// TIA Portal project "VISU_Umsetzer+Sauggreifer_Template" (V14)

(* hardware
DEVICE "S7300/ET200M-Station_1"  S7-300 station
   slot 0: "Profilschiene_0"  Rail  6ES7 390-1***0-0AA0
   slot 2: "PLC_1"  CPU 315-2 PN/DP  6ES7 315-2EH13-0AB0  V2.6
      slot 1: "MPI/DP-Schnittstelle_1"  X1
      slot 2: "PROFINET-Schnittstelle_1"  PN-IO
         slot 1: "Port_1"  Port
*)

// ===== PLC "PLC_1"  CPU 315-2 PN/DP =====

VAR_GLOBAL   // PLC tag table "Standard-Variablentabelle"
   "POS_X_PLUS" AT %I10.3 : Bool;   // Greifer bei Position X+
   "POS_X_MIDDLE" AT %I10.4 : Bool;   // Greifer bei Position X Mitte
   "POS_X_MINUS" AT %I10.5 : Bool;   // Greifer bei Position X-
   "POS_Z_PLUS" AT %I10.6 : Bool;   // Greifer bei Position Z+
   "POS_Z_MINUS" AT %I10.7 : Bool;   // Greifer bei Position Z-
   "STORAGE_ENGAGED" AT %I11.0 : Bool;   // Ablageplatz belegt
   "BELT1_ENGAGED" AT %I11.3 : Bool;   // Förderband 1 belegt
   "BELT2_ENGAGED" AT %I11.4 : Bool;   // Förderband 2 belegt
   "TO_X_PLUS" AT %Q4.0 : Bool;   // Greifer nach X+ fahren
   "TO_X_MINUS" AT %Q4.1 : Bool;   // Greifer nach X- fahren
   "TO_Z_PLUS" AT %Q4.2 : Bool;   // Greifer nach Z+ fahren
   "TO_Z_MINUS" AT %Q4.3 : Bool;   // Greifer nach Z- fahren
   "BELT1_TO_X_PLUS" AT %Q4.4 : Bool;   // Förderband 1 nach X+
   "BELT1_TO_X_MINUS" AT %Q4.5 : Bool;   // Förderband 1 nach X-
   "BELT2_TO_X_PLUS" AT %Q4.6 : Bool;   // Förderband 2 nach X+
   "BELT2_TO_X_MINUS" AT %Q4.7 : Bool;   // Förderband 2 nach X-
   "PUMP_ON" AT %Q5.0 : Bool;   // Greiferpumpe an
   "CONTROL_KEY_1" AT %I11.1 : Bool;   // Bedientaster 1
   "CONTROL_KEY_2" AT %I11.2 : Bool;   // Bedientaster 2
   "INIT_0" AT %M0.0 : Bool;   // 1 - Initschritt 0 abgeschlossen
   "INIT_1" AT %M0.1 : Bool;   // 1 - Initschritt 1 abgeschlossen
   "INIT_2" AT %M0.2 : Bool;   // 1 - Initschritt 2 abgeschlossen
   "STEP" AT %MW2 : Int;
   "RESET(1)" AT %M1.6 : Bool;
   "Trig_ContrKey1" AT %M0.3 : Bool;   // 1 - Pos Flanke
   "Trig_Step_1" AT %M0.6 : Bool;   // 1 - Pos Flanke
   "Trig_ContrKey2" AT %M0.4 : Bool;   // 1 - Pos Flanke
   "STORAGE" AT %M1.3 : Bool;   // 1 - Ablage zu Belt 2
   "Trig_Step_2" AT %M0.7 : Bool;   // 1 - Pos Flanke
   "BELT1_BELT2" AT %M1.2 : Bool;
   "BELT1_STORAGE" AT %M1.1 : Bool;
   "Trig_Step_3" AT %M1.0 : Bool;   // 1 - Pos Flanke
   "INC_CHN_A" AT %I10.0 : Bool;   // Inkrementalgeber X-Achse Kanal A
   "INC_CHN_B" AT %I10.1 : Bool;   // Inkrementalgeber X-Achse Kanal B
   "INC_CHN_Z" AT %I10.2 : Bool;   // Inkrementalgeber X-Achse Kanal C
   "X_POSITION" AT %MD1000 : DInt;   // X-Position Greifer
   "Trig_Chan_A" AT %M1.5 : Bool;   // 1 - Pos Flanke
   "Trig_Chan_B" AT %M1.4 : Bool;   // 1 - Pos Flanke
   "INTERN" AT %MW6 : Int;
   "D_INTERN" AT %MD8 : DInt;
END_VAR

DATA_BLOCK "Incremental_DB"   // DB2
{ S7_Optimized_Access := 'FALSE' }
VERSION : 0.1
// stored: InstanceOfName Incremental
"Incremental"
BEGIN
END_DATA_BLOCK

FUNCTION_BLOCK "Incremental"   // FB1, FBD
{ S7_Optimized_Access := 'FALSE' }
VERSION : 0.1
   VAR_INPUT
      KANAL_A : Bool;
      KANAL_B : Bool;
      RESET : Bool;
   END_VAR
   VAR_OUTPUT
      Number : DInt;
   END_VAR
   VAR_TEMP   // added for the SCL form of the ladder/FBD networks
      _w1 : Bool;
   END_VAR
BEGIN

REGION Network 1
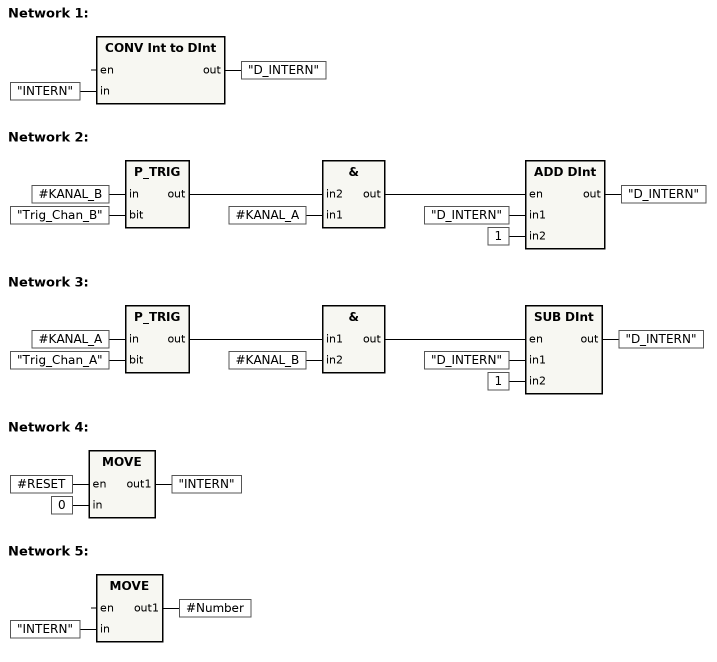
   "D_INTERN" := INT_TO_DINT("INTERN");
END_REGION

REGION Network 2
   #_w1 := #KANAL_B AND NOT "Trig_Chan_B";   // rising edge
   "Trig_Chan_B" := #KANAL_B;
   IF #_w1 AND #KANAL_A THEN "D_INTERN" := "D_INTERN" + 1; END_IF;
END_REGION

REGION Network 3
   #_w1 := #KANAL_A AND NOT "Trig_Chan_A";   // rising edge
   "Trig_Chan_A" := #KANAL_A;
   IF #_w1 AND #KANAL_B THEN "D_INTERN" := "D_INTERN" - 1; END_IF;
END_REGION

REGION Network 4
   IF #RESET THEN "INTERN" := 0; END_IF;
END_REGION

REGION Network 5
   #Number := "INTERN";
END_REGION
END_FUNCTION_BLOCK

ORGANIZATION_BLOCK "Main"   // OB1, FBD
TITLE = "Main Program Sweep (Cycle)"
{ S7_Optimized_Access := 'FALSE' }
VERSION : 0.1
   VAR_TEMP
      OB1_EV_CLASS : Byte;   // Bits 0-3 = 1 (Coming event), Bits 4-7 = 1 (Event class 1)
      OB1_SCAN_1 : Byte;   // 1 (Cold restart scan 1 of OB 1), 3 (Scan 2-n of OB 1)
      OB1_PRIORITY : Byte;   // Priority of OB Execution
      OB1_OB_NUMBR : Byte;   // 1 (Organization block 1, OB1)
      OB1_RESERVED_1 : Byte;   // Reserved for system
      OB1_RESERVED_2 : Byte;   // Reserved for system
      OB1_PREV_CYCLE : Int;   // Cycle time of previous OB1 scan (milliseconds)
      OB1_MIN_CYCLE : Int;   // Minimum cycle time of OB1 (milliseconds)
      OB1_MAX_CYCLE : Int;   // Maximum cycle time of OB1 (milliseconds)
      OB1_DATE_TIME : Date_And_Time;   // Date and time OB1 started
   END_VAR
   VAR_TEMP   // added for the SCL form of the ladder/FBD networks
      _w1 : Bool;
      _w2 : Bool;
   END_VAR
BEGIN

REGION Network 1: Initialisierung - Z hoch
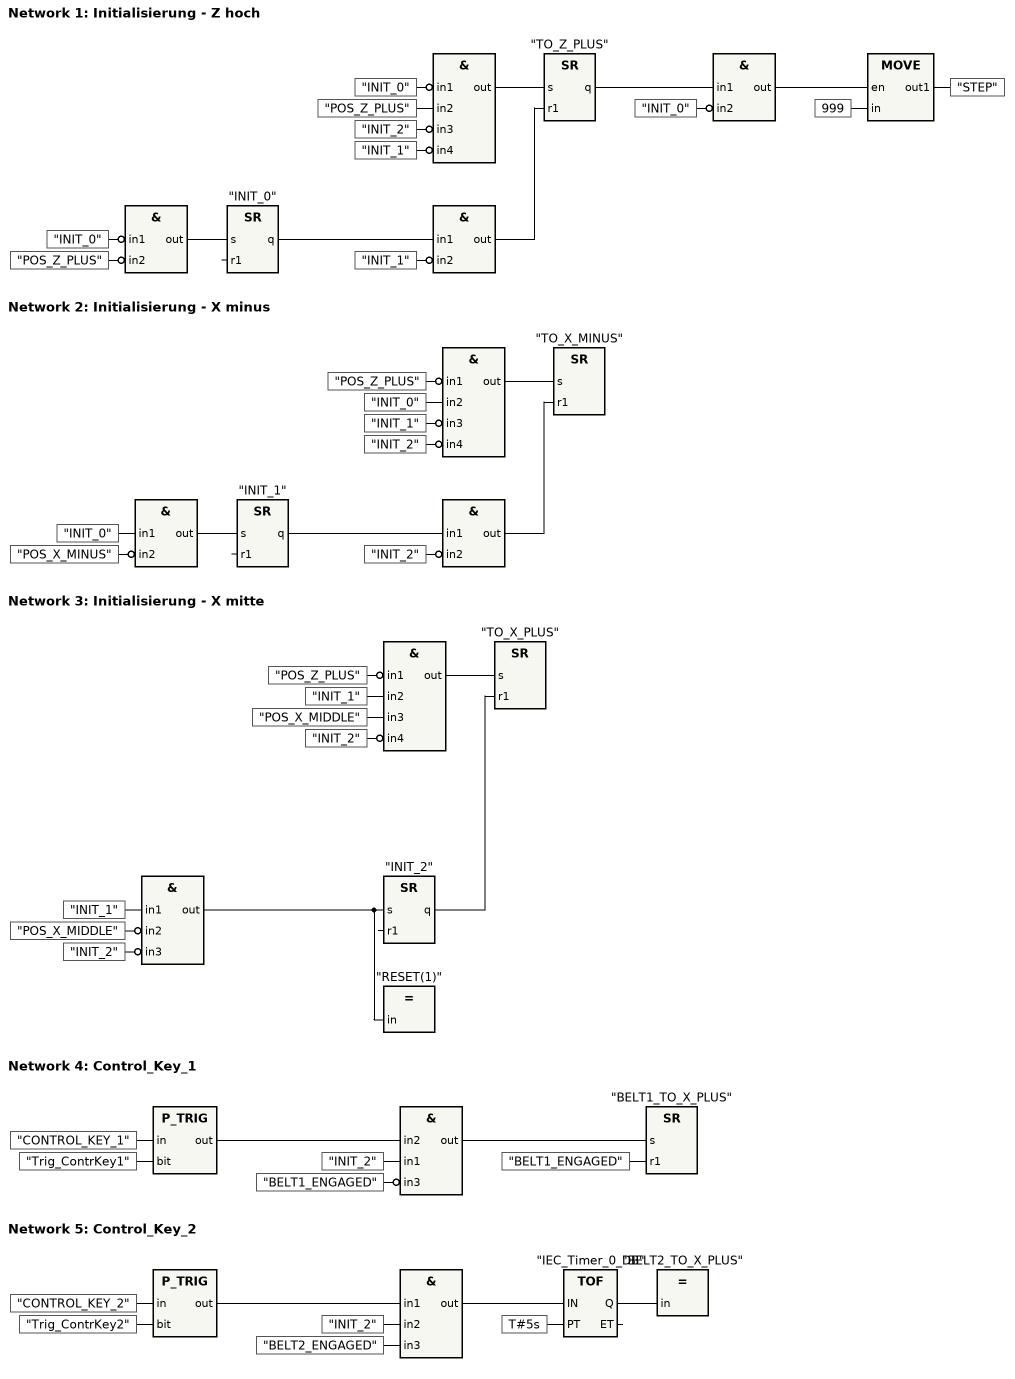
   #_w1 := NOT "INIT_0" AND "POS_Z_PLUS" AND NOT "INIT_2" AND NOT "INIT_1";
   IF NOT "INIT_0" AND NOT "POS_Z_PLUS" THEN
       "INIT_0" := TRUE;   // SR flip-flop
   END_IF;
   IF #_w1 THEN
       "TO_Z_PLUS" := TRUE;   // SR flip-flop
   END_IF;
   IF "INIT_0" AND NOT "INIT_1" THEN "TO_Z_PLUS" := FALSE; END_IF;
   IF "TO_Z_PLUS" AND NOT "INIT_0" THEN "STEP" := 999; END_IF;
END_REGION

REGION Network 2: Initialisierung - X minus
   #_w1 := NOT "POS_Z_PLUS" AND "INIT_0" AND NOT "INIT_1" AND NOT "INIT_2";
   IF "INIT_0" AND NOT "POS_X_MINUS" THEN
       "INIT_1" := TRUE;   // SR flip-flop
   END_IF;
   IF #_w1 THEN
       "TO_X_MINUS" := TRUE;   // SR flip-flop
   END_IF;
   IF "INIT_1" AND NOT "INIT_2" THEN "TO_X_MINUS" := FALSE; END_IF;
END_REGION

REGION Network 3: Initialisierung - X mitte
   #_w1 := "INIT_1" AND NOT "POS_X_MIDDLE" AND NOT "INIT_2";
   #_w2 := NOT "POS_Z_PLUS" AND "INIT_1" AND "POS_X_MIDDLE" AND NOT "INIT_2";
   IF #_w1 THEN
       "INIT_2" := TRUE;   // SR flip-flop
   END_IF;
   IF #_w2 THEN
       "TO_X_PLUS" := TRUE;   // SR flip-flop
   END_IF;
   IF "INIT_2" THEN "TO_X_PLUS" := FALSE; END_IF;
   "RESET(1)" := #_w1;
END_REGION

REGION Network 4: Control_Key_1
   #_w1 := "CONTROL_KEY_1" AND NOT "Trig_ContrKey1";   // rising edge
   "Trig_ContrKey1" := "CONTROL_KEY_1";
   IF #_w1 AND "INIT_2" AND NOT "BELT1_ENGAGED" THEN
       "BELT1_TO_X_PLUS" := TRUE;   // SR flip-flop
   END_IF;
   IF "BELT1_ENGAGED" THEN "BELT1_TO_X_PLUS" := FALSE; END_IF;
END_REGION

REGION Network 5: Control_Key_2
   #_w1 := "CONTROL_KEY_2" AND NOT "Trig_ContrKey2";   // rising edge
   "Trig_ContrKey2" := "CONTROL_KEY_2";
   "IEC_Timer_0_DB".TOF(IN := #_w1 AND "INIT_2" AND "BELT2_ENGAGED", PT := T#5s);
   "BELT2_TO_X_PLUS" := "IEC_Timer_0_DB".Q;
END_REGION

REGION Network 6: Storage räumen
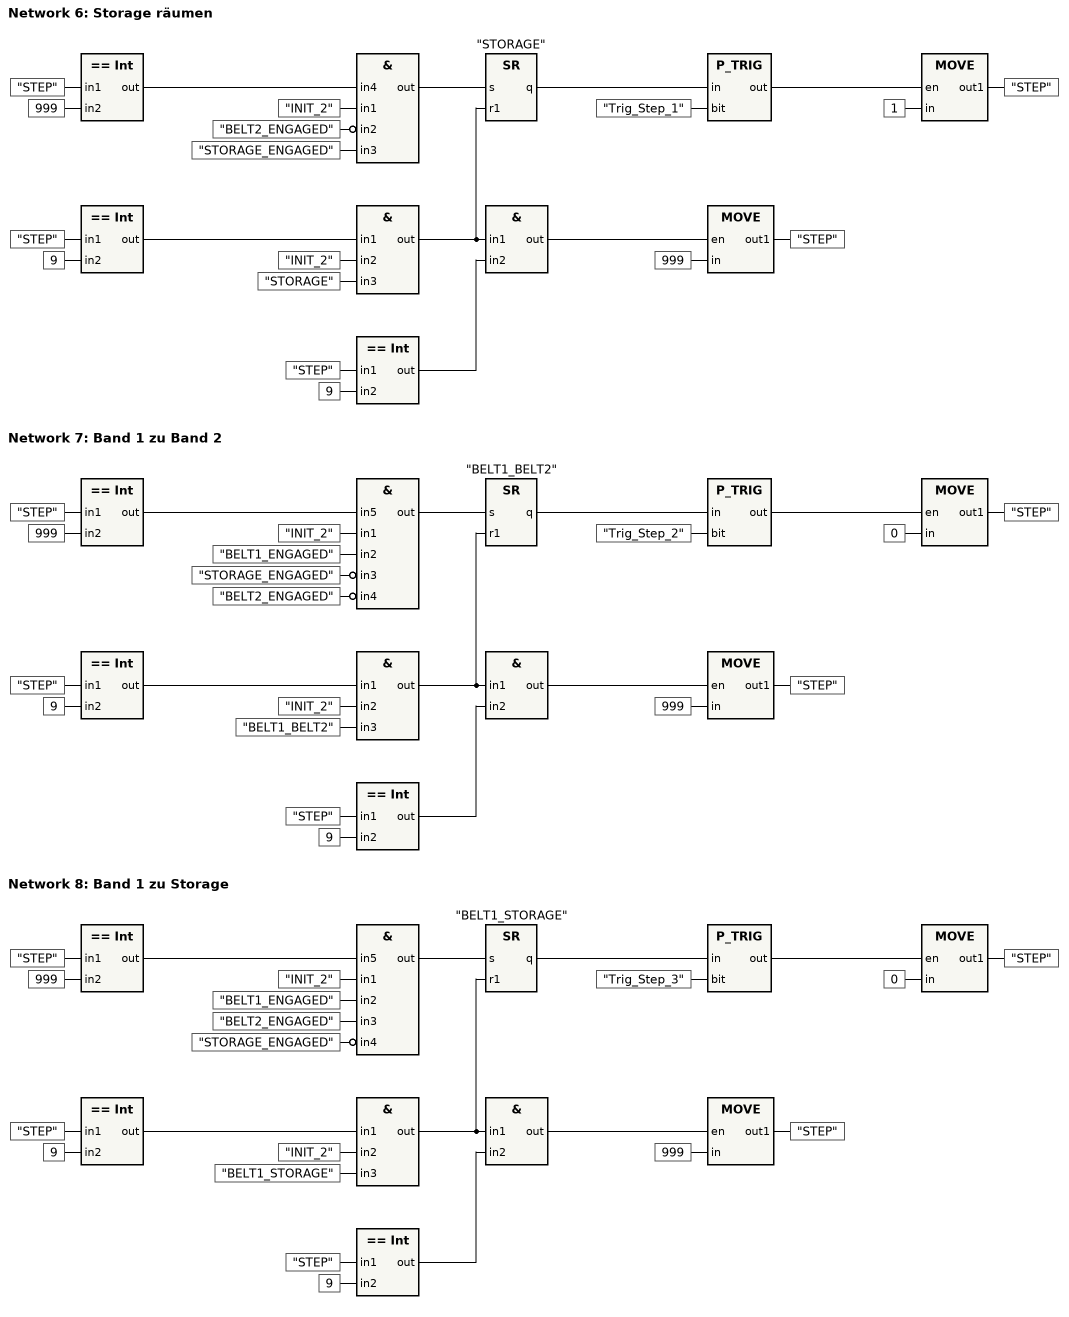
   #_w1 := ("STEP" = 9) AND "INIT_2" AND "STORAGE";
   IF ("STEP" = 999) AND "INIT_2" AND NOT "BELT2_ENGAGED" AND "STORAGE_ENGAGED" THEN
       "STORAGE" := TRUE;   // SR flip-flop
   END_IF;
   IF #_w1 THEN "STORAGE" := FALSE; END_IF;
   #_w2 := "STORAGE" AND NOT "Trig_Step_1";   // rising edge
   "Trig_Step_1" := "STORAGE";
   IF #_w2 THEN "STEP" := 1; END_IF;
   IF #_w1 AND ("STEP" = 9) THEN "STEP" := 999; END_IF;
END_REGION

REGION Network 7: Band 1 zu Band 2
   #_w1 := ("STEP" = 9) AND "INIT_2" AND "BELT1_BELT2";
   IF ("STEP" = 999) AND "INIT_2" AND "BELT1_ENGAGED" AND NOT "STORAGE_ENGAGED" AND NOT "BELT2_ENGAGED" THEN
       "BELT1_BELT2" := TRUE;   // SR flip-flop
   END_IF;
   IF #_w1 THEN "BELT1_BELT2" := FALSE; END_IF;
   #_w2 := "BELT1_BELT2" AND NOT "Trig_Step_2";   // rising edge
   "Trig_Step_2" := "BELT1_BELT2";
   IF #_w2 THEN "STEP" := 0; END_IF;
   IF #_w1 AND ("STEP" = 9) THEN "STEP" := 999; END_IF;
END_REGION

REGION Network 8: Band 1 zu Storage
   #_w1 := ("STEP" = 9) AND "INIT_2" AND "BELT1_STORAGE";
   IF ("STEP" = 999) AND "INIT_2" AND "BELT1_ENGAGED" AND "BELT2_ENGAGED" AND NOT "STORAGE_ENGAGED" THEN
       "BELT1_STORAGE" := TRUE;   // SR flip-flop
   END_IF;
   IF #_w1 THEN "BELT1_STORAGE" := FALSE; END_IF;
   #_w2 := "BELT1_STORAGE" AND NOT "Trig_Step_3";   // rising edge
   "Trig_Step_3" := "BELT1_STORAGE";
   IF #_w2 THEN "STEP" := 0; END_IF;
   IF #_w1 AND ("STEP" = 9) THEN "STEP" := 999; END_IF;
END_REGION

REGION Network 9: x minus
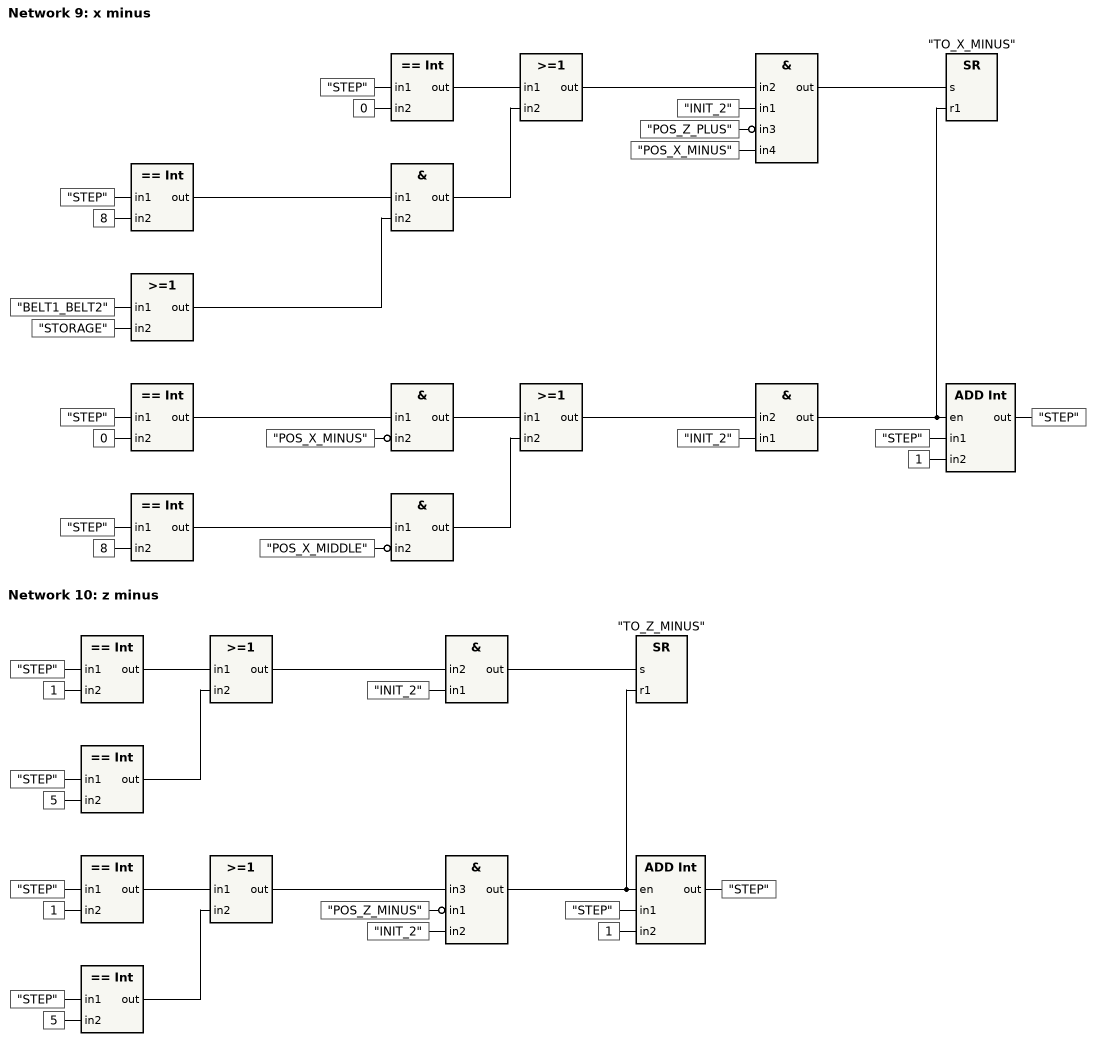
   #_w1 := ((("STEP" = 0) AND NOT "POS_X_MINUS") OR (("STEP" = 8) AND NOT "POS_X_MIDDLE")) AND "INIT_2";
   IF (("STEP" = 0) OR (("STEP" = 8) AND ("BELT1_BELT2" OR "STORAGE"))) AND "INIT_2" AND NOT "POS_Z_PLUS" AND "POS_X_MINUS" THEN
       "TO_X_MINUS" := TRUE;   // SR flip-flop
   END_IF;
   IF #_w1 THEN
       "TO_X_MINUS" := FALSE;
       "STEP" := "STEP" + 1;
   END_IF;
END_REGION

REGION Network 10: z minus
   #_w1 := (("STEP" = 1) OR ("STEP" = 5)) AND NOT "POS_Z_MINUS" AND "INIT_2";
   IF (("STEP" = 1) OR ("STEP" = 5)) AND "INIT_2" THEN
       "TO_Z_MINUS" := TRUE;   // SR flip-flop
   END_IF;
   IF #_w1 THEN
       "TO_Z_MINUS" := FALSE;
       "STEP" := "STEP" + 1;
   END_IF;
END_REGION

REGION Network 11: saug an
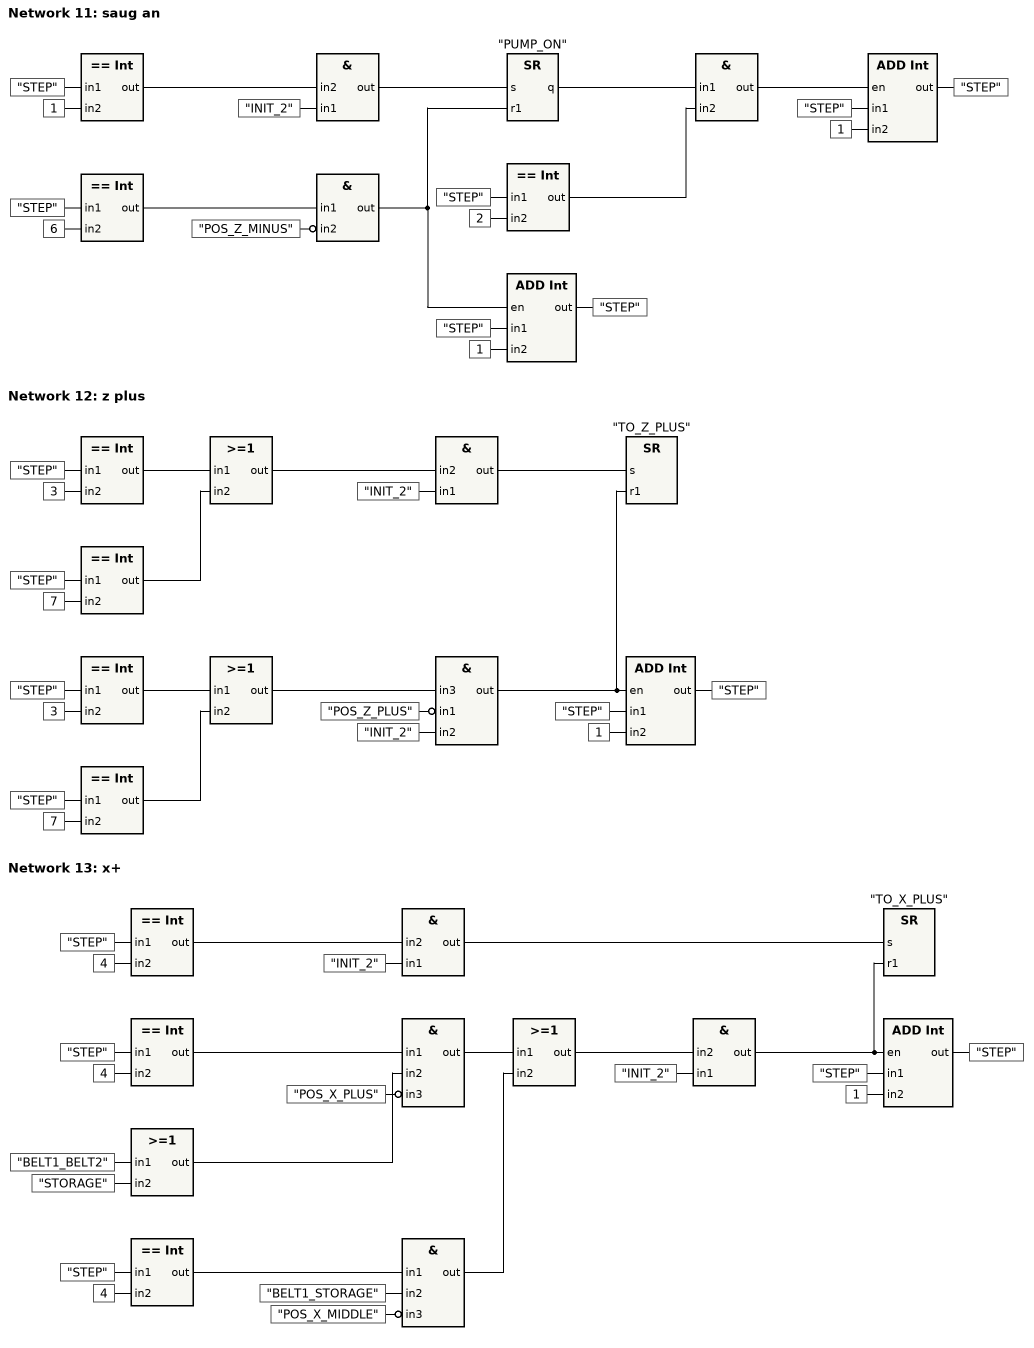
   #_w1 := ("STEP" = 6) AND NOT "POS_Z_MINUS";
   IF ("STEP" = 1) AND "INIT_2" THEN
       "PUMP_ON" := TRUE;   // SR flip-flop
   END_IF;
   IF #_w1 THEN "PUMP_ON" := FALSE; END_IF;
   IF "PUMP_ON" AND ("STEP" = 2) THEN "STEP" := "STEP" + 1; END_IF;
   IF #_w1 THEN "STEP" := "STEP" + 1; END_IF;
END_REGION

REGION Network 12: z plus
   #_w1 := (("STEP" = 3) OR ("STEP" = 7)) AND NOT "POS_Z_PLUS" AND "INIT_2";
   IF (("STEP" = 3) OR ("STEP" = 7)) AND "INIT_2" THEN
       "TO_Z_PLUS" := TRUE;   // SR flip-flop
   END_IF;
   IF #_w1 THEN
       "TO_Z_PLUS" := FALSE;
       "STEP" := "STEP" + 1;
   END_IF;
END_REGION

REGION Network 13: x+
   #_w1 := ((("STEP" = 4) AND ("BELT1_BELT2" OR "STORAGE") AND NOT "POS_X_PLUS") OR (("STEP" = 4) AND "BELT1_STORAGE" AND NOT "POS_X_MIDDLE")) AND "INIT_2";
   IF ("STEP" = 4) AND "INIT_2" THEN
       "TO_X_PLUS" := TRUE;   // SR flip-flop
   END_IF;
   IF #_w1 THEN
       "TO_X_PLUS" := FALSE;
       "STEP" := "STEP" + 1;
   END_IF;
END_REGION

REGION Network 14
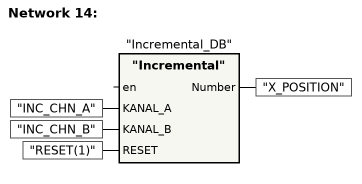
   "Incremental_DB"(KANAL_A := "INC_CHN_A", KANAL_B := "INC_CHN_B", RESET := "RESET(1)", Number => "X_POSITION");   // "Incremental"
END_REGION
END_ORGANIZATION_BLOCK